// Mitsubishi GX Works2 project: projectPLC_Group9   PLC: FX3G

// global labels: Global1
VAR_GLOBAL
  Start_day_Button AT X007 : BOOL;
  End_day AT M1 : BOOL;
  Working_day AT M2 : BOOL;
  Out_of_stock AT M3 : BOOL;
  Emergency_button AT X005 : BOOL;
  Working_day_light AT Y000 : BOOL;
  Insert_stock AT M4 : BOOL;
  Oat_input AT D1112 : REAL;
  Protein_input AT D1106 : REAL;
  Honey_input AT D1120 : REAL;
  Honey_stock AT D1102 : REAL;
  Oat_stock AT D1130 : REAL;
  Protein_stock AT D1118 : REAL;
  Analog_output AT D8282 : INT;
  Total_storage AT D1100 : REAL;
  Choose_bar AT X003 : BOOL;
END_VAR
VAR_GLOBAL CONSTANT
  Min_amount : REAL := 400;
  Min_amount_honey : REAL := 120;
  Min_amount_oat : REAL := 240;
  Min_amount_protein : REAL := 160;
END_VAR
VAR_GLOBAL
  Out_of_stock_classic AT M5 : BOOL;
  Is_out_of_stock AT M6 : BOOL;
  start_Working_day AT M2 : BOOL;
  Out_of_stock_Protein AT M7 : BOOL;
END_VAR
VAR_GLOBAL CONSTANT
  Min_amount_oat_c : REAL := 400;
  Min_amount_honey_c : REAL := 120;
  Min_amount_protein_c : REAL := 160;
  Min_amount_oat_p : REAL := 240;
  Min_amount_honey_p : REAL := 160;
  Min_amount_protein_p : REAL := 320;
END_VAR
VAR_GLOBAL
  Choose_Type_Analog AT D8280 : INT;
END_VAR
VAR_GLOBAL CONSTANT
  Convert : INT := 400;
END_VAR
VAR_GLOBAL
  Chosen_Type_0_10 AT D1200 : REAL;
  Make_Classic AT M9 : BOOL;
END_VAR
VAR_GLOBAL CONSTANT
  Choose_classic : REAL := 5;
END_VAR
VAR_GLOBAL
  Make_protein AT M8 : BOOL;
END_VAR
VAR_GLOBAL CONSTANT
  Timer_5sec : INT := 50;
END_VAR
VAR_GLOBAL
  Start_Mix AT TC1 : BOOL;
  Finish_Mix AT TS1 : BOOL;
  Mix_light AT Y003 : BOOL;
  Classic_container AT D1500 : REAL;
  Protein_Container AT D1600 : REAL;
  insert_analog AT D8054 : INT;
  insert_analog3 AT D7033 : REAL;
  Baking_light AT X002 : BOOL;
  Baking_Button AT X002 : BOOL;
  Baking_Classic AT TC5 : BOOL;
END_VAR
VAR_GLOBAL CONSTANT
  Timer_4sec_Classic : INT := 40;
END_VAR
VAR_GLOBAL
  Baking_Protein AT TC6 : BOOL;
END_VAR
VAR_GLOBAL CONSTANT
  Timer_5sec_Protein : WORD := 50;
END_VAR
VAR_GLOBAL
  Baking_Classic_Finished AT TS5 : BOOL;
  Baking_Protein_Finished AT TS6 : BOOL;
  Baking_Finished AT M20 : BOOL;
  Baking_Timer AT TC8 : BOOL;
END_VAR
VAR_GLOBAL CONSTANT
  Flashing_light : INT := 1;
END_VAR
VAR_GLOBAL
  Baking_Timer_Finished AT TS8 : BOOL;
  First_light AT Y001 : BOOL;
  Baking_Timer2 AT TC9 : BOOL;
  Second_Light AT Y002 : BOOL;
  Baking_Timer2_Finished AT TS9 : BOOL;
  Baking_process AT M21 : BOOL;
  Packing_finished AT M12 : BOOL;
  Start_storage AT X006 : BOOL;
  Pack_Bar AT X000 : BOOL;
  Counter_packing AT CC1 : BOOL;
END_VAR
VAR_GLOBAL CONSTANT
  Bars : INT := 8;
  Starting_Point : INT;
END_VAR
VAR_GLOBAL
  Packed_Bars AT CN1 : INT;
  New_Package AT M25 : BOOL;
  First_bar_lamp AT Y004 : BOOL;
  Counter_packing_Finished AT CS1 : BOOL;
  Mix_is_finished AT M28 : BOOL;
  Storage AT D2024 : INT;
END_VAR
VAR_GLOBAL CONSTANT
  add_one : INT := 1;
END_VAR
VAR_GLOBAL
  Error AT M24 : BOOL;
END_VAR
VAR_GLOBAL CONSTANT
  divide_by_ten : INT := 10;
END_VAR
VAR_GLOBAL
  Flash_help AT M35 : BOOL;
  finish_classic_bake AT M34 : BOOL;
  finish_protein_bake AT M38 : BOOL;
  Saved_choice AT D7033 : REAL;
END_VAR
VAR_GLOBAL CONSTANT
  Eight_Bars : INT := 8;
END_VAR
VAR_GLOBAL
  Indicator_light AT M26 : BOOL;
END_VAR
VAR_GLOBAL CONSTANT
  Zero : INT;
  Analog_DIV : REAL := 40;
END_VAR
VAR_GLOBAL
  Number_of_packs AT D1135 : REAL;
END_VAR

// task Task_01 (event TRUE, interval 0, priority 31): POU_01

PROGRAM POU_01
(* structured ladder/FBD written out as ST: instructions are called as NAME(EN, inputs, outputs); _pN, _eN, _tN stand for wires *)
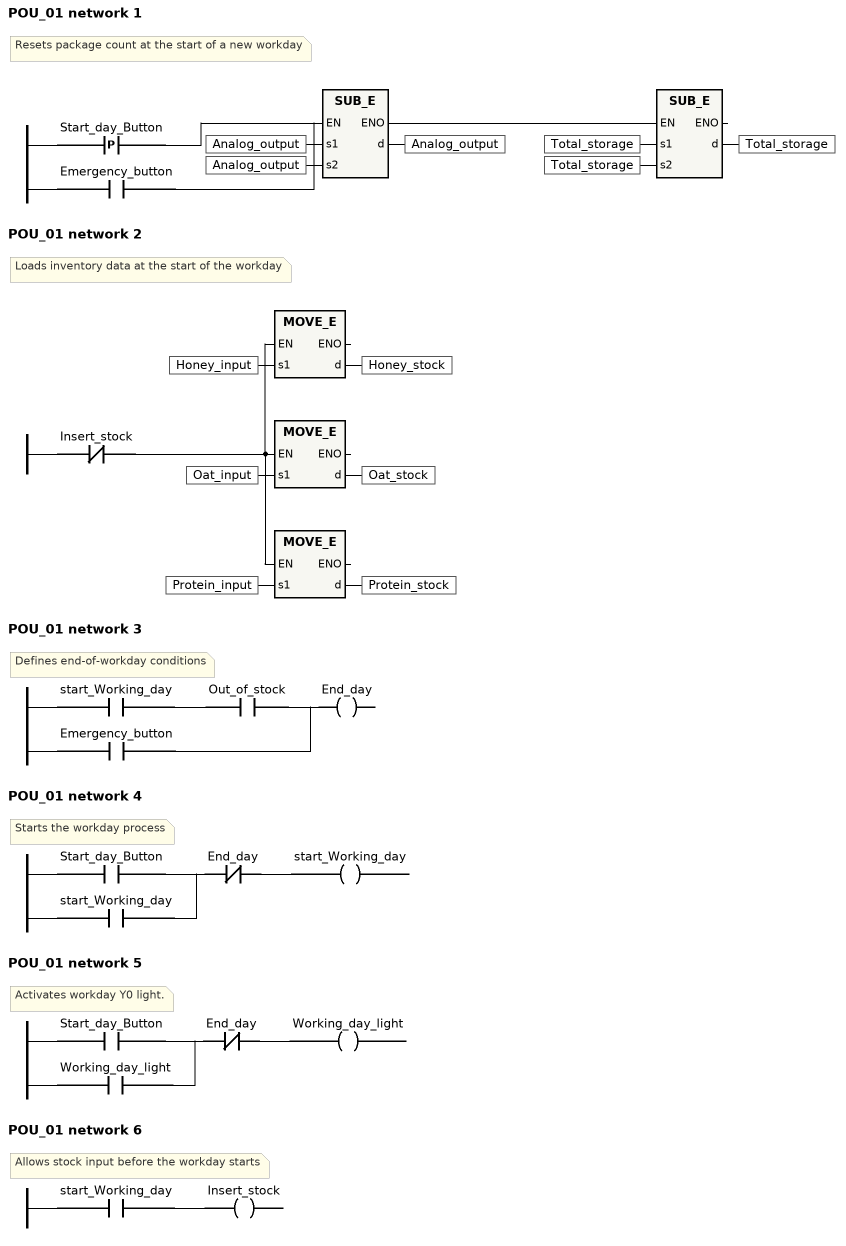
(* network 1 *)
(* Resets package count at the start of a new workday *)
_e1 := SUB_E(LDP(TRUE, Start_day_Button) OR Emergency_button, Analog_output, Analog_output, Analog_output);
SUB_E(_e1, Total_storage, Total_storage, Total_storage);
(* network 2 *)
(* Loads inventory data at the start of the workday *)
_p1 := NOT Insert_stock;
MOVE_E(_p1, Honey_input, Honey_stock);
MOVE_E(_p1, Oat_input, Oat_stock);
MOVE_E(_p1, Protein_input, Protein_stock);
(* network 3 *)
(* Defines end-of-workday conditions *)
End_day := (start_Working_day AND Out_of_stock) OR Emergency_button;
(* network 4 *)
(* Starts the workday process *)
start_Working_day := (Start_day_Button OR start_Working_day) AND NOT End_day;
(* network 5 *)
(* Activates workday Y0 light. *)
Working_day_light := (Start_day_Button OR Working_day_light) AND NOT End_day;
(* network 6 *)
(* Allows stock input before the workday starts *)
Insert_stock := start_Working_day;
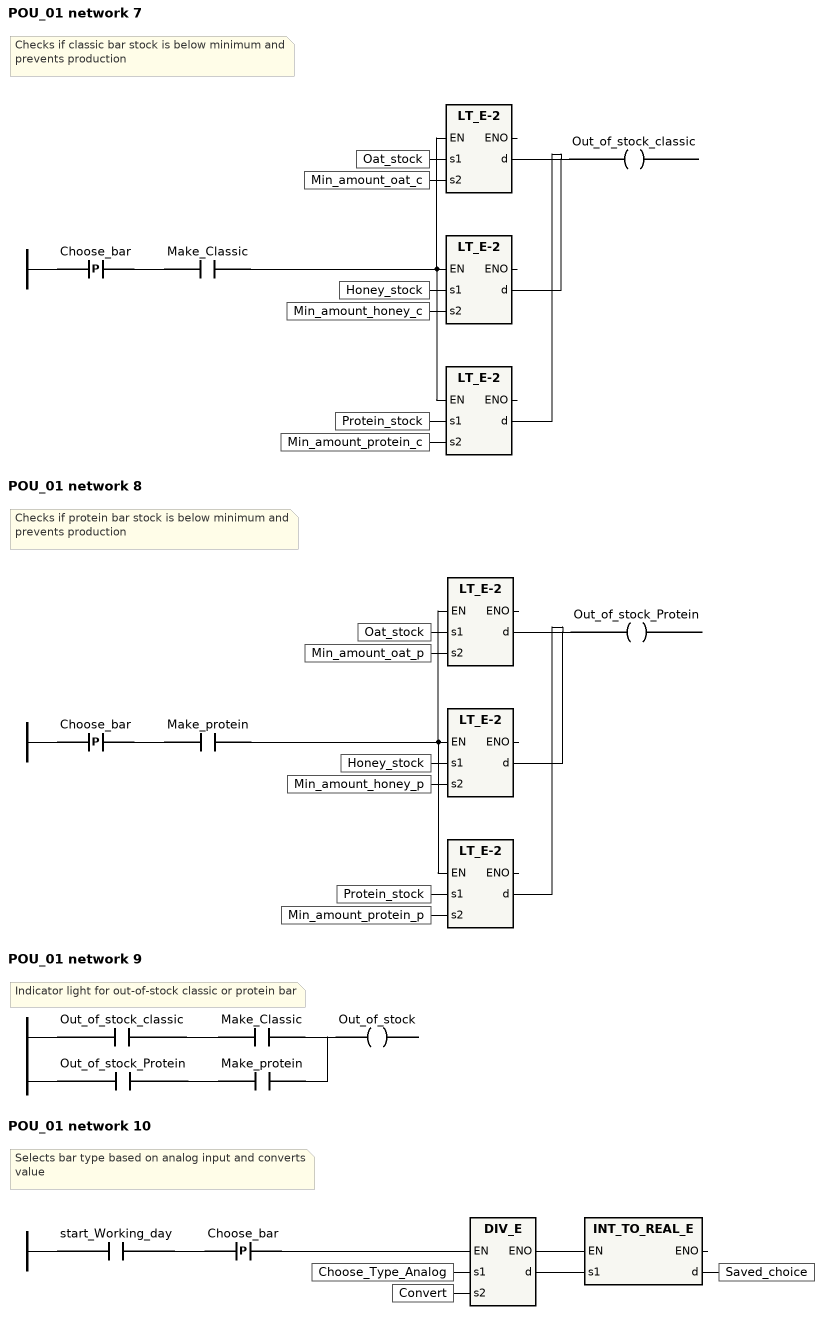
(* network 7 *)
(* Checks if classic bar stock is below minimum and prevents production *)
_p1 := LDP(TRUE, Choose_bar) AND Make_Classic;
LT_E(_p1, Oat_stock, Min_amount_oat_c, _t2);
LT_E(_p1, Honey_stock, Min_amount_honey_c, _t3);
LT_E(_p1, Protein_stock, Min_amount_protein_c, _t4);
Out_of_stock_classic := _t2 OR _t3 OR _t4;
(* network 8 *)
(* Checks if protein bar stock is below minimum and prevents production *)
_p1 := LDP(TRUE, Choose_bar) AND Make_protein;
LT_E(_p1, Oat_stock, Min_amount_oat_p, _t2);
LT_E(_p1, Honey_stock, Min_amount_honey_p, _t3);
LT_E(_p1, Protein_stock, Min_amount_protein_p, _t4);
Out_of_stock_Protein := _t2 OR _t3 OR _t4;
(* network 9 *)
(* Indicator light for out-of-stock classic or protein bar *)
Out_of_stock := (Out_of_stock_classic AND Make_Classic) OR (Out_of_stock_Protein AND Make_protein);
(* network 10 *)
(* Selects bar type based on analog input and converts value *)
_e2 := DIV_E(start_Working_day AND LDP(TRUE, Choose_bar), Choose_Type_Analog, Convert, _t1);
INT_TO_REAL_E(_e2, _t1, Saved_choice);
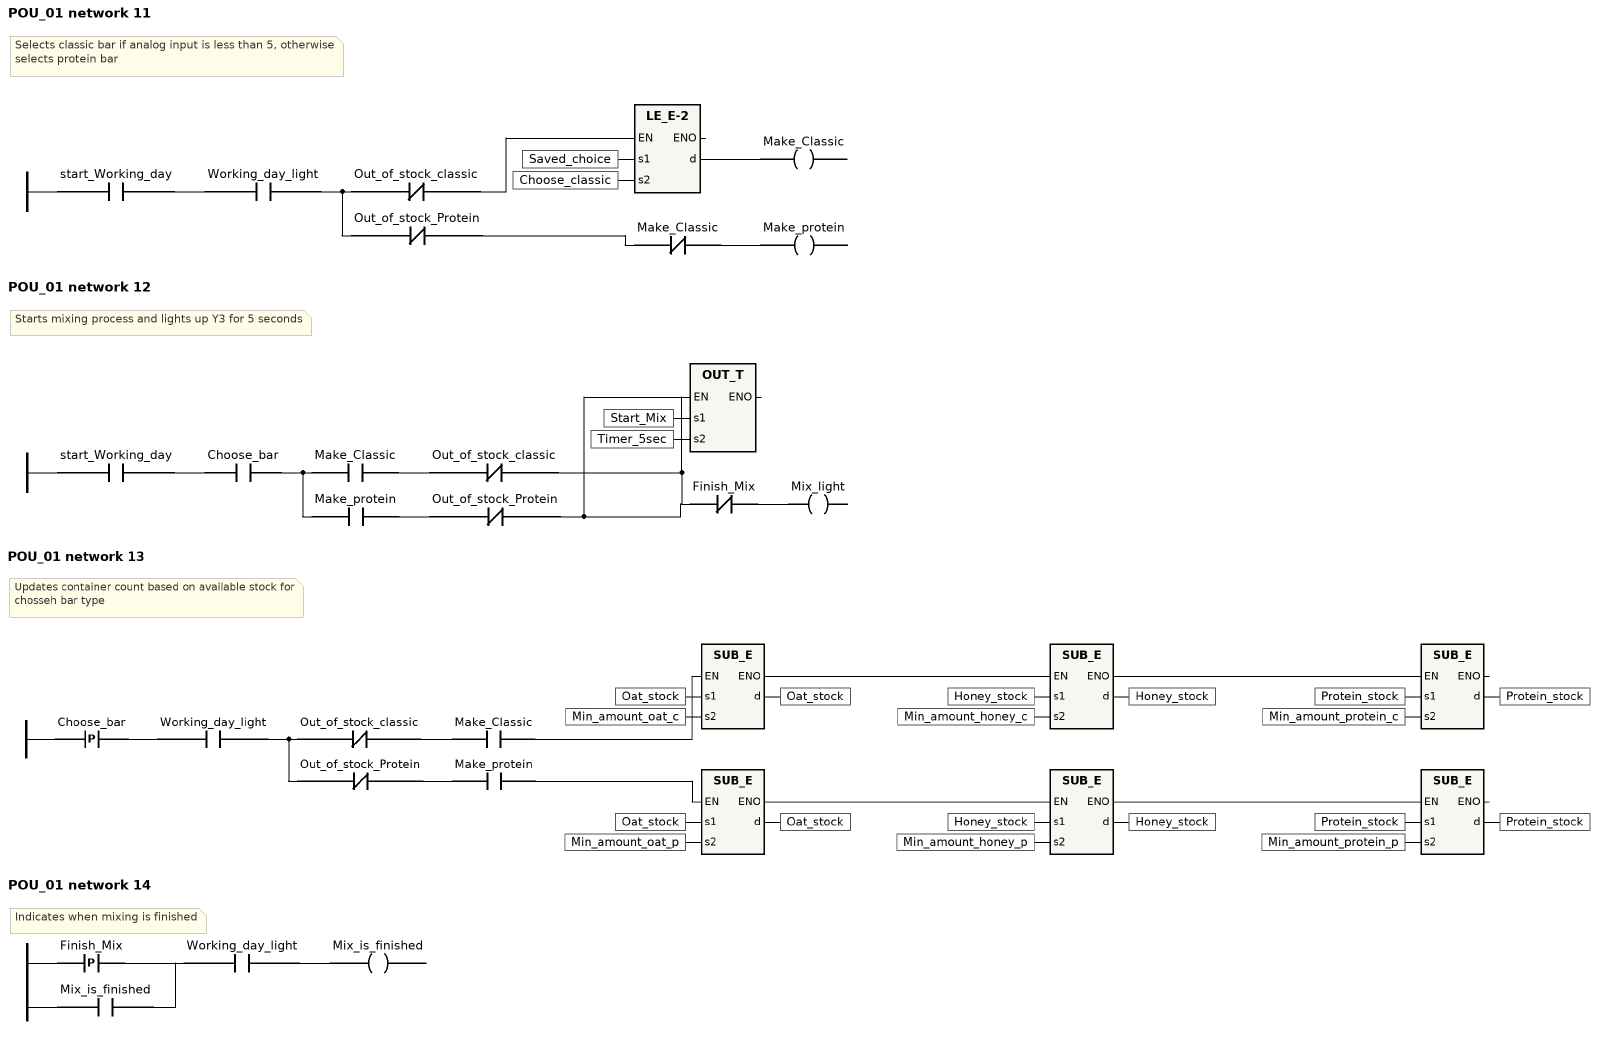
(* network 11 *)
(* Selects classic bar if analog input is less than 5, otherwise selects protein bar *)
_p1 := start_Working_day AND Working_day_light;
LE_E(_p1 AND NOT Out_of_stock_classic, Saved_choice, Choose_classic, _t2);
Make_Classic := _t2;
Make_protein := _p1 AND NOT Out_of_stock_Protein AND NOT Make_Classic;
(* network 12 *)
(* Starts mixing process and lights up Y3 for 5 seconds *)
_p1 := start_Working_day AND Choose_bar;
_p2 := (_p1 AND Make_Classic AND NOT Out_of_stock_classic) OR (_p1 AND Make_protein AND NOT Out_of_stock_Protein);
OUT_T(_p2, Start_Mix, Timer_5sec);
Mix_light := _p2 AND NOT Finish_Mix;
(* network 13 *)
(* Updates container count based on available stock for chosseh bar type *)
_p1 := LDP(TRUE, Choose_bar) AND Working_day_light;
_e2 := SUB_E(_p1 AND NOT Out_of_stock_classic AND Make_Classic, Oat_stock, Min_amount_oat_c, Oat_stock);
_e3 := SUB_E(_e2, Honey_stock, Min_amount_honey_c, Honey_stock);
SUB_E(_e3, Protein_stock, Min_amount_protein_c, Protein_stock);
_e4 := SUB_E(_p1 AND NOT Out_of_stock_Protein AND Make_protein, Oat_stock, Min_amount_oat_p, Oat_stock);
_e5 := SUB_E(_e4, Honey_stock, Min_amount_honey_p, Honey_stock);
SUB_E(_e5, Protein_stock, Min_amount_protein_p, Protein_stock);
(* network 14 *)
(* Indicates when mixing is finished *)
Mix_is_finished := (LDP(TRUE, Finish_Mix) OR Mix_is_finished) AND Working_day_light;
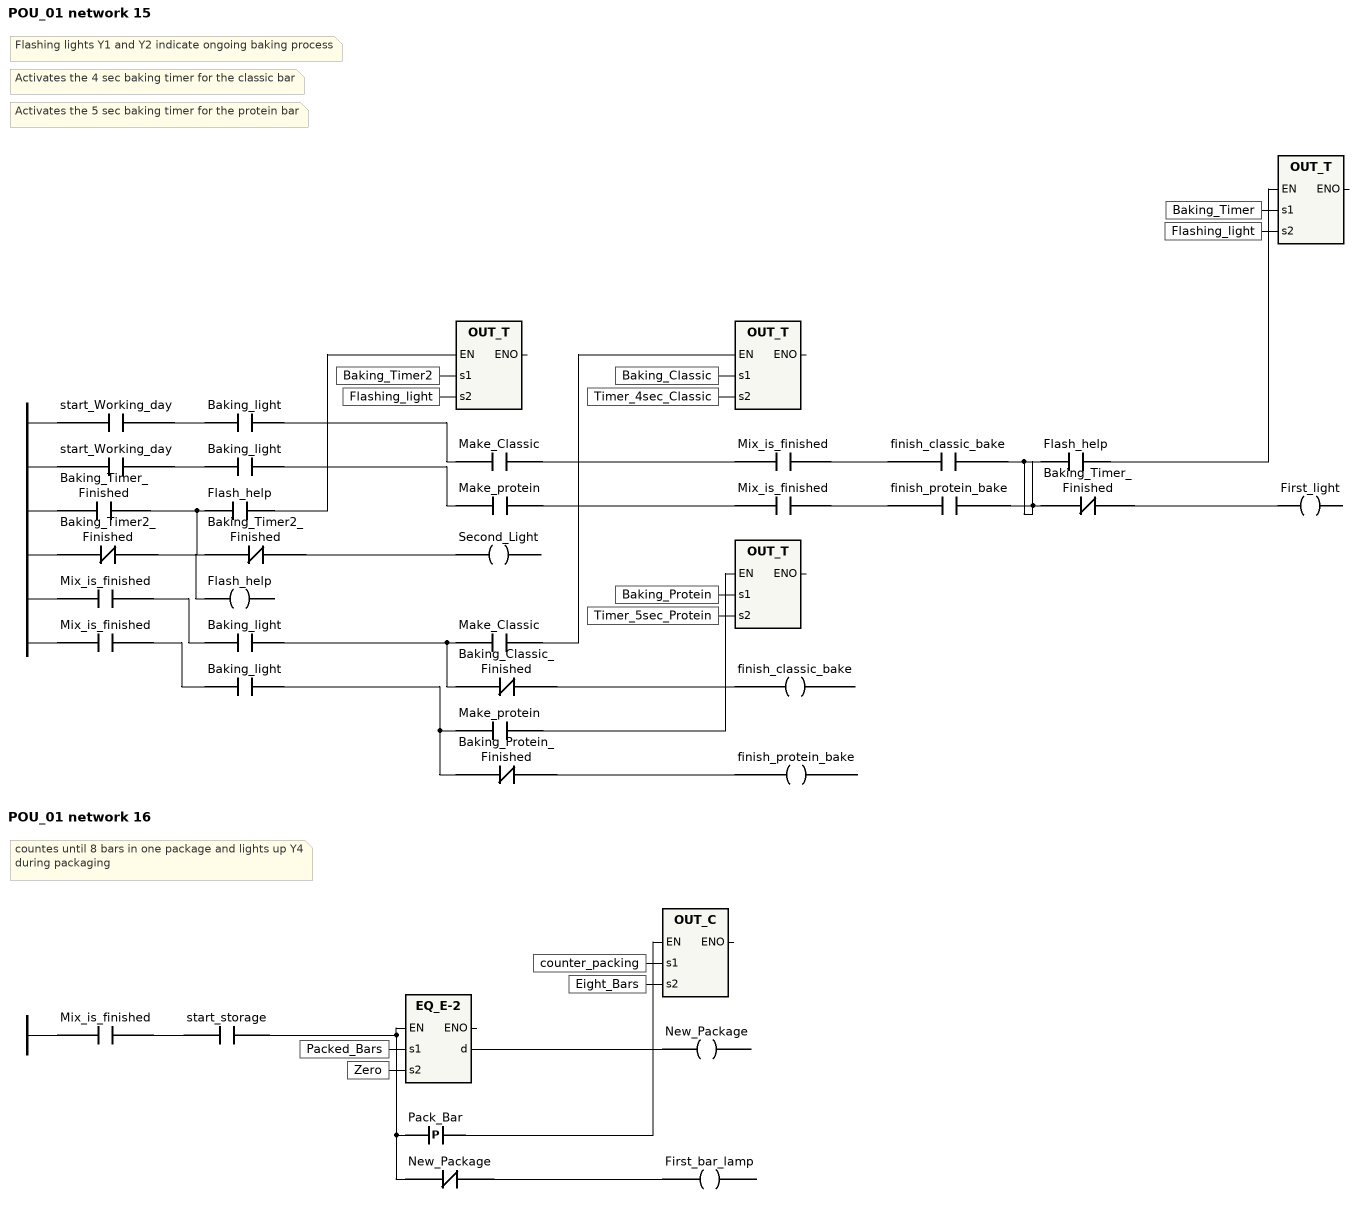
(* network 15 *)
(* Flashing lights Y1 and Y2 indicate ongoing baking process *)
(* Activates the 4 sec baking timer for the classic bar *)
(* Activates the 5 sec baking timer for the protein bar *)
_p1 := (start_Working_day AND Baking_light AND Make_Classic AND Mix_is_finished AND finish_classic_bake) OR (start_Working_day AND Baking_light AND Make_protein AND Mix_is_finished AND finish_protein_bake);
OUT_T(_p1 AND Flash_help, Baking_Timer, Flashing_light);
First_light := _p1 AND NOT Baking_Timer_Finished;
OUT_T(Baking_Timer_Finished AND Flash_help, Baking_Timer2, Flashing_light);
Second_Light := Baking_Timer_Finished AND NOT Baking_Timer2_Finished;
Flash_help := NOT Baking_Timer2_Finished;
_p2 := Mix_is_finished AND Baking_light;
OUT_T(_p2 AND Make_Classic, Baking_Classic, Timer_4sec_Classic);
finish_classic_bake := _p2 AND NOT Baking_Classic_Finished;
_p3 := Mix_is_finished AND Baking_light;
OUT_T(_p3 AND Make_protein, Baking_Protein, Timer_5sec_Protein);
finish_protein_bake := _p3 AND NOT Baking_Protein_Finished;
(* network 16 *)
(* countes until 8 bars in one package and lights up Y4 during packaging *)
_p1 := Mix_is_finished AND start_storage;
OUT_C(_p1 AND LDP(TRUE, Pack_Bar), counter_packing, Eight_Bars);
EQ_E(_p1, Packed_Bars, Zero, _t2);
New_Package := _t2;
First_bar_lamp := _p1 AND NOT New_Package;
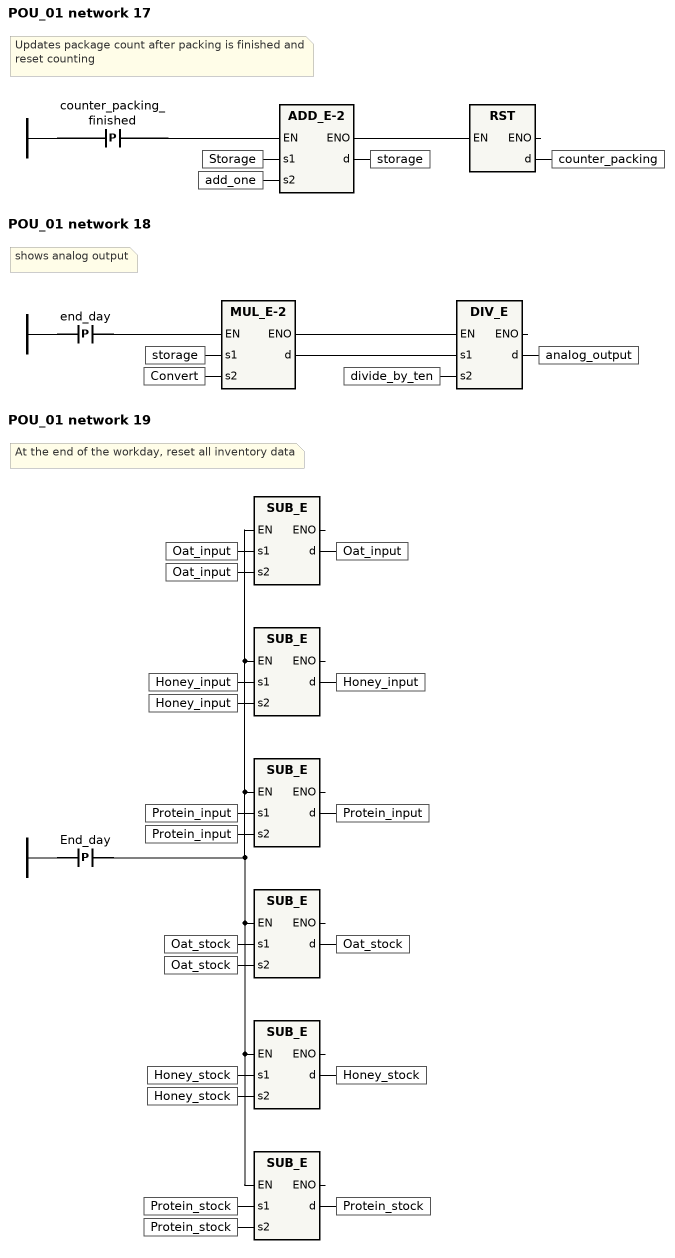
(* network 17 *)
(* Updates package count after packing is finished and reset counting *)
_e1 := ADD_E(LDP(TRUE, counter_packing_finished), Storage, add_one, storage);
RST(_e1, counter_packing);
(* network 18 *)
(* shows analog output *)
_e2 := MUL_E(LDP(TRUE, end_day), storage, Convert, _t1);
DIV_E(_e2, _t1, divide_by_ten, analog_output);
(* network 19 *)
(* At the end of the workday, reset all inventory data *)
_p1 := LDP(TRUE, End_day);
SUB_E(_p1, Oat_input, Oat_input, Oat_input);
SUB_E(_p1, Honey_input, Honey_input, Honey_input);
SUB_E(_p1, Protein_input, Protein_input, Protein_input);
SUB_E(_p1, Oat_stock, Oat_stock, Oat_stock);
SUB_E(_p1, Honey_stock, Honey_stock, Honey_stock);
SUB_E(_p1, Protein_stock, Protein_stock, Protein_stock);
END_PROGRAM
